// TIA Portal V20 export
// export: Created 2025-12-01T14:56:13.6216389Z, ExportSetting None, DisplayName Totally Integrated Automation Portal, DisplayVersion V20 Update 3, DisplayName TIA Portal Openness, DisplayVersion V20 Update 3, DisplayName TIA Portal Version Control Interface, DisplayVersion V20 Update 3, DisplayName STEP 7 Professional, DisplayVersion V20 Update 3, DisplayName STEP 7 Safety, DisplayVersion V20 Update 2, DisplayName WinCC Basic/Comfort/Advanced, DisplayVersion V20 Update 3, DisplayName WinCC Professional, DisplayVersion V20 Update 3, DisplayName WinCC Unified, DisplayVersion V20 Update 3
TYPE "UDT_EstadoZonaDispositivo"
   STRUCT
      Pulsador { S7_SetPoint := 'True'} : "PulsadorZona";
      Estado { S7_SetPoint := 'True'} : "EstadoZona";   // Estado de la Zona
      CodigoError : UDInt;   // Codigo de Error de la Zona
      VariablesInternas { S7_SetPoint := 'True'} : "InternasDeLaZona";   // Variables internas y sinoptico
   END_STRUCT;
   // Pulsador.P_Auto := false;
END_TYPE
